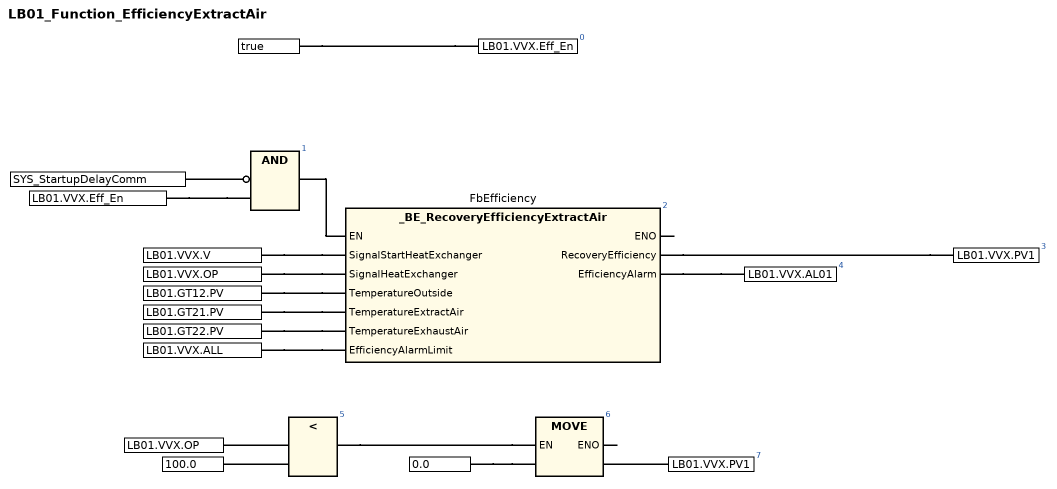
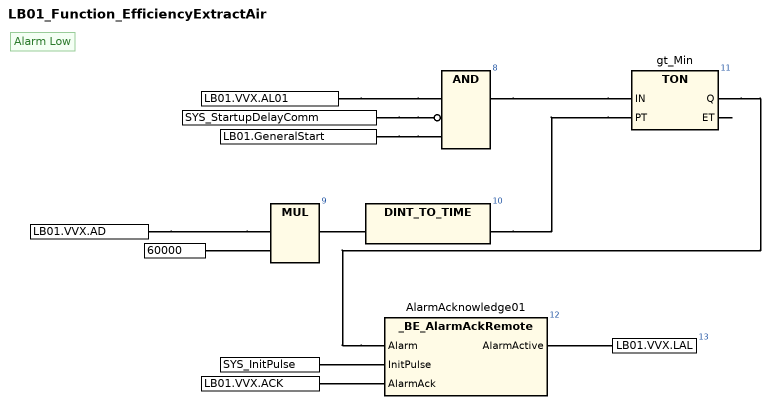
LB01.VVX.Eff_En := true;
IF NOT SYS_StartupDelayComm AND LB01.VVX.Eff_En THEN
    FbEfficiency(
        SignalStartHeatExchanger := LB01.VVX.V,
        SignalHeatExchanger := LB01.VVX.OP,
        TemperatureOutside := LB01.GT12.PV,
        TemperatureExtractAir := LB01.GT21.PV,
        TemperatureExhaustAir := LB01.GT22.PV,
        EfficiencyAlarmLimit := LB01.VVX.ALL); // _BE_RecoveryEfficiencyExtractAir
END_IF
LB01.VVX.PV1 := FbEfficiency.RecoveryEfficiency;
LB01.VVX.AL01 := FbEfficiency.EfficiencyAlarm;
IF LB01.VVX.OP < 100.0 THEN _w1 := 0.0; END_IF
LB01.VVX.PV1 := _w1;
// Alarm Low
gt_Min(IN := LB01.VVX.AL01 AND NOT SYS_StartupDelayComm AND LB01.GeneralStart, PT := DINT_TO_TIME(LB01.VVX.AD * 60000)); // TON
AlarmAcknowledge01(Alarm := gt_Min.Q, InitPulse := SYS_InitPulse, AlarmAck := LB01.VVX.ACK); // _BE_AlarmAckRemote
LB01.VVX.LAL := AlarmAcknowledge01.AlarmActive;

END_PROGRAM

// Device/AREA1/B001/LB01/Function/LB01_Function_Overtime
PROGRAM LB01_Function_Overtime
VAR
	FbOvertime: _BE_OverTime;
END_VAR

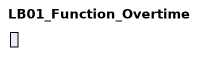
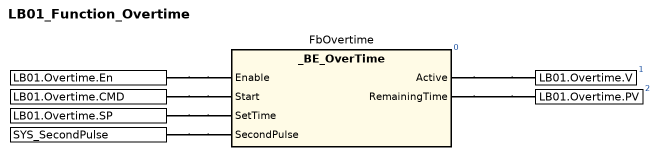
FbOvertime(
    Enable := LB01.Overtime.En,
    Start := LB01.Overtime.CMD,
    SetTime := LB01.Overtime.SP,
    SecondPulse := SYS_SecondPulse); // _BE_OverTime
LB01.Overtime.V := FbOvertime.Active;
LB01.Overtime.PV := FbOvertime.RemainingTime;

END_PROGRAM

// Device/AREA1/B001/LB01/Function/LB01_Function_Preheating
PROGRAM LB01_Function_Preheating
VAR
	plsGeneralStart: BOOL;
	plsStart: R_TRIG;
	delayStartControl: TON;
END_VAR
VAR // added by the converter: edge detectors and wires of the graphical bodies
    _w1, _w3, _w4 : ANY;
    _w2 : BOOL;
END_VAR

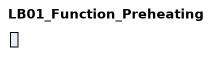
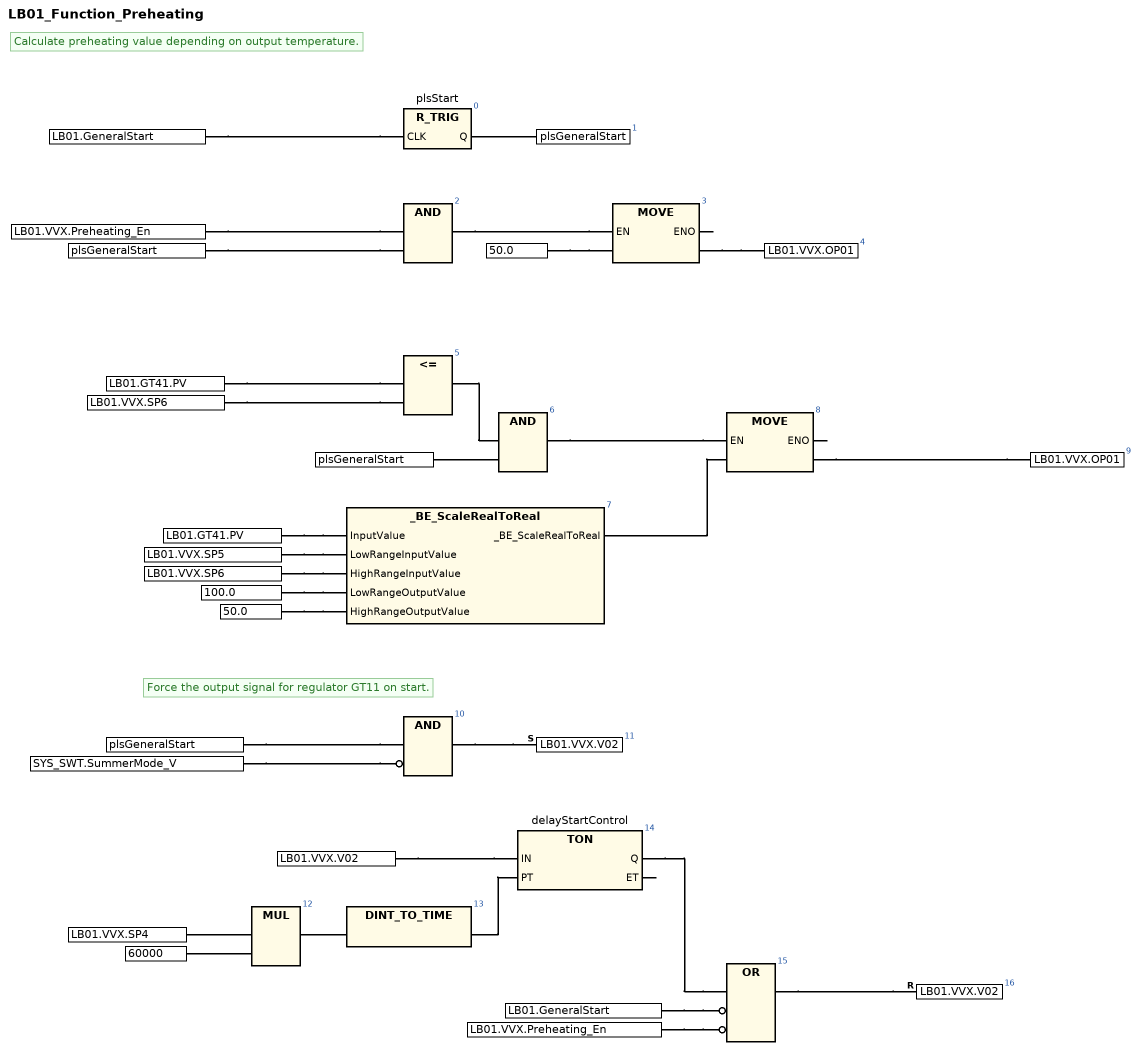
// Calculate preheating value depending on output temperature.
plsStart(CLK := LB01.GeneralStart); // R_TRIG
plsGeneralStart := plsStart.Q;
IF LB01.VVX.Preheating_En AND plsGeneralStart THEN _w1 := 50.0; END_IF
LB01.VVX.OP01 := _w1;
_w2 := LB01.GT41.PV <= LB01.VVX.SP6 AND plsGeneralStart;
_w3 := _BE_ScaleRealToReal(InputValue := LB01.GT41.PV, LowRangeInputValue := LB01.VVX.SP5, HighRangeInputValue := LB01.VVX.SP6, LowRangeOutputValue := 100.0, HighRangeOutputValue := 50.0);
IF _w2 THEN _w4 := _w3; END_IF
LB01.VVX.OP01 := _w4;
// Force the output signal for regulator GT11 on start.
LB01.VVX.V02 S= plsGeneralStart AND NOT SYS_SWT.SummerMode_V;
delayStartControl(IN := LB01.VVX.V02, PT := DINT_TO_TIME(LB01.VVX.SP4 * 60000)); // TON
LB01.VVX.V02 R= delayStartControl.Q OR NOT LB01.GeneralStart OR NOT LB01.VVX.Preheating_En;

END_PROGRAM

// Device/AREA1/B001/LB01/Sensor/Humidity/GM21/LB01_GM21
PROGRAM LB01_GM21
VAR
	local:strSensor7_Humidity;
	gt_Min: TON;
	gt_Max: TON;
	reset_en: RS;
	ackLal: BOOL;
	ackHal: BOOL;
	AlarmAcknowledge01: _BE_AlarmAckRemote;
	AlarmAcknowledge02: _BE_AlarmAckRemote;
END_VAR
VAR // added by the converter: edge detectors and wires of the graphical bodies
    _w1, _w3, _w4 : ANY;
    _w2 : BOOL;
END_VAR

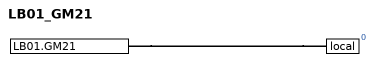
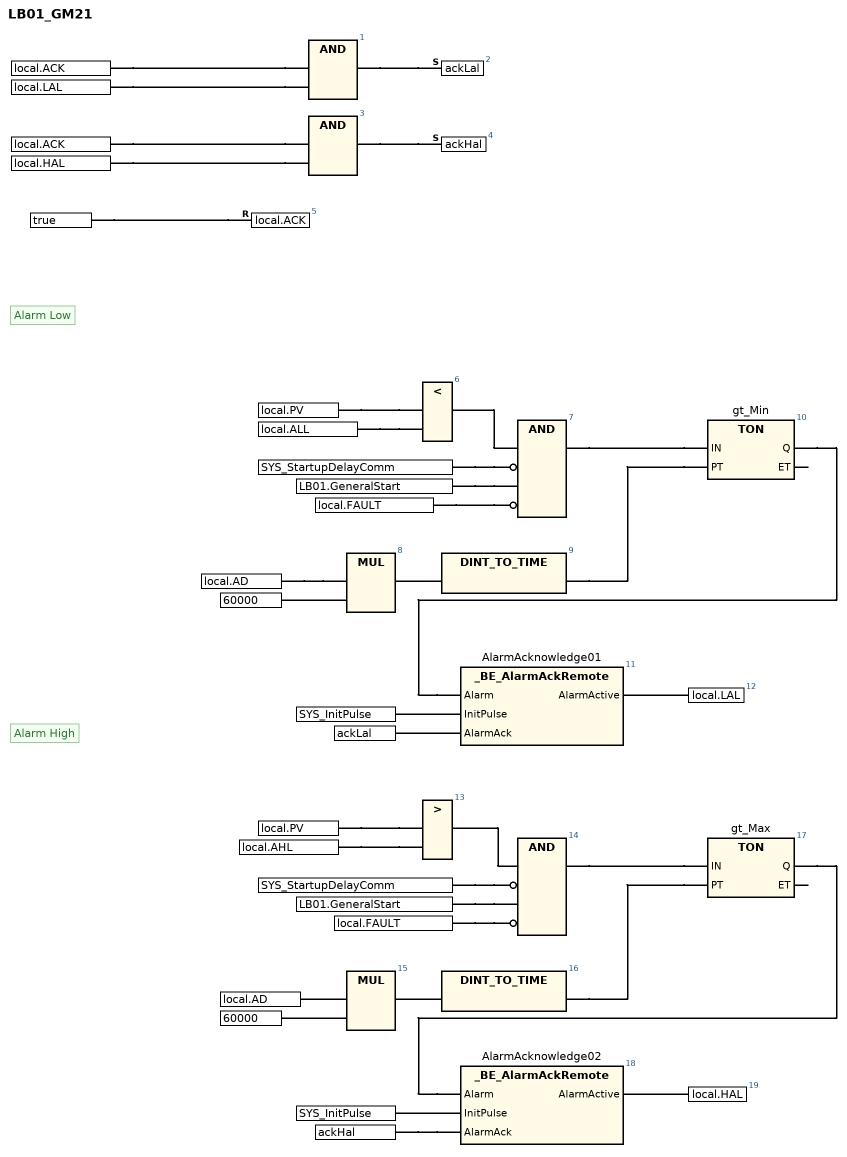
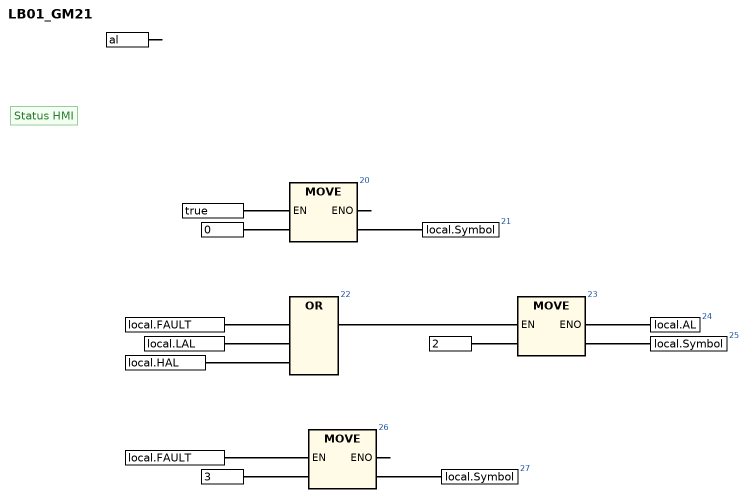
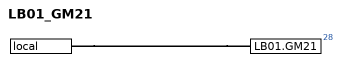
// note: 4 stored wires end on pins the file does not list and are not shown
local := LB01.GM21;
ackLal S= local.ACK AND local.LAL;
ackHal S= local.ACK AND local.HAL;
local.ACK R= true;
// Alarm Low
gt_Min(IN := local.PV < local.ALL AND NOT SYS_StartupDelayComm AND LB01.GeneralStart AND NOT local.FAULT, PT := DINT_TO_TIME(local.AD * 60000)); // TON
AlarmAcknowledge01(Alarm := gt_Min.Q, InitPulse := SYS_InitPulse, AlarmAck := ackLal); // _BE_AlarmAckRemote
local.LAL := AlarmAcknowledge01.AlarmActive;
// Alarm High
gt_Max(IN := local.PV > local.AHL AND NOT SYS_StartupDelayComm AND LB01.GeneralStart AND NOT local.FAULT, PT := DINT_TO_TIME(local.AD * 60000)); // TON
AlarmAcknowledge02(Alarm := gt_Max.Q, InitPulse := SYS_InitPulse, AlarmAck := ackHal); // _BE_AlarmAckRemote
local.HAL := AlarmAcknowledge02.AlarmActive;
// Status HMI
IF true THEN _w1 := 0; END_IF
local.Symbol := _w1;
_w2 := local.FAULT OR local.LAL OR local.HAL;
IF _w2 THEN _w3 := 2; END_IF
local.AL := _w2;
local.Symbol := _w3;
IF local.FAULT THEN _w4 := 3; END_IF
local.Symbol := _w4;
LB01.GM21 := local;
// al: input not connected

END_PROGRAM

// Device/AREA1/B001/LB01/Function/LB01_NightCooling
PROGRAM LB01_NightCooling
VAR
	fbNightCool: _BE_NightCooling;
END_VAR

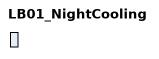
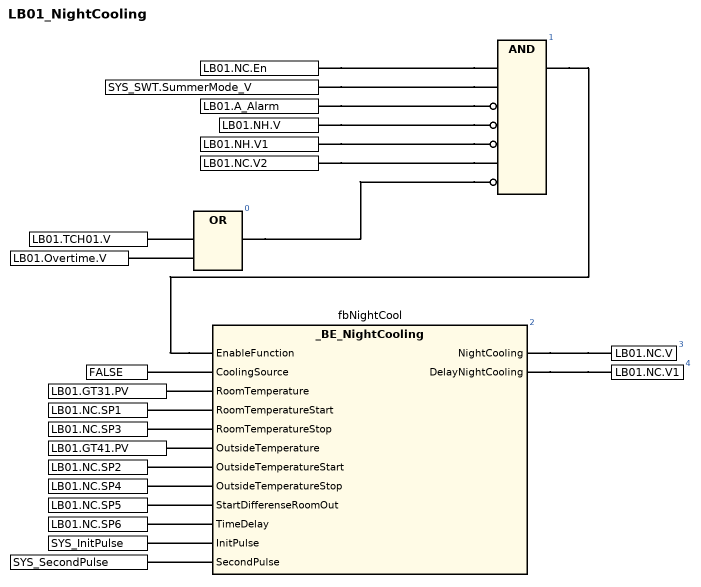
fbNightCool(
    EnableFunction := LB01.NC.En AND SYS_SWT.SummerMode_V AND NOT LB01.A_Alarm AND NOT LB01.NH.V AND NOT LB01.NH.V1 AND LB01.NC.V2 AND NOT (LB01.TCH01.V OR LB01.Overtime.V),
    CoolingSource := FALSE,
    RoomTemperature := LB01.GT31.PV,
    RoomTemperatureStart := LB01.NC.SP1,
    RoomTemperatureStop := LB01.NC.SP3,
    OutsideTemperature := LB01.GT41.PV,
    OutsideTemperatureStart := LB01.NC.SP2,
    OutsideTemperatureStop := LB01.NC.SP4,
    StartDifferenseRoomOut := LB01.NC.SP5,
    TimeDelay := LB01.NC.SP6,
    InitPulse := SYS_InitPulse,
    SecondPulse := SYS_SecondPulse); // _BE_NightCooling
LB01.NC.V := fbNightCool.NightCooling;
LB01.NC.V1 := fbNightCool.DelayNightCooling;

END_PROGRAM

// Device/AREA1/B001/LB01/Function/LB01_NightHeating
PROGRAM LB01_NightHeating
VAR
	fbNightHeat: _BE_NightHeating;
END_VAR

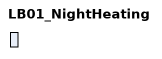
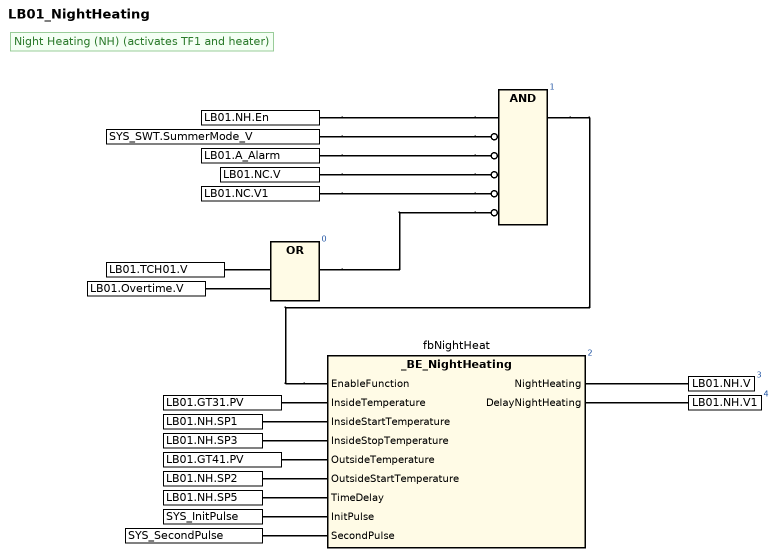
// Night Heating (NH) (activates TF1 and heater)
fbNightHeat(
    EnableFunction := LB01.NH.En AND NOT SYS_SWT.SummerMode_V AND NOT LB01.A_Alarm AND NOT LB01.NC.V AND NOT LB01.NC.V1 AND NOT (LB01.TCH01.V OR LB01.Overtime.V),
    InsideTemperature := LB01.GT31.PV,
    InsideStartTemperature := LB01.NH.SP1,
    InsideStopTemperature := LB01.NH.SP3,
    OutsideTemperature := LB01.GT41.PV,
    OutsideStartTemperature := LB01.NH.SP2,
    TimeDelay := LB01.NH.SP5,
    InitPulse := SYS_InitPulse,
    SecondPulse := SYS_SecondPulse); // _BE_NightHeating
LB01.NH.V := fbNightHeat.NightHeating;
LB01.NH.V1 := fbNightHeat.DelayNightHeating;

END_PROGRAM

// Device/AREA1/B001/UC/Sh1/Alarms/UCSh1_Alarms
PROGRAM UCSh1_Alarms
VAR
	AlarmAcknowledge01: _BE_AlarmAckRemote;
	timerManMode: TON;
	_BE_AlarmAckRemote_0: _BE_AlarmAckRemote;
END_VAR
VAR // added by the converter: edge detectors and wires of the graphical bodies
    _w1 : BOOL;
END_VAR

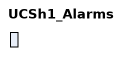
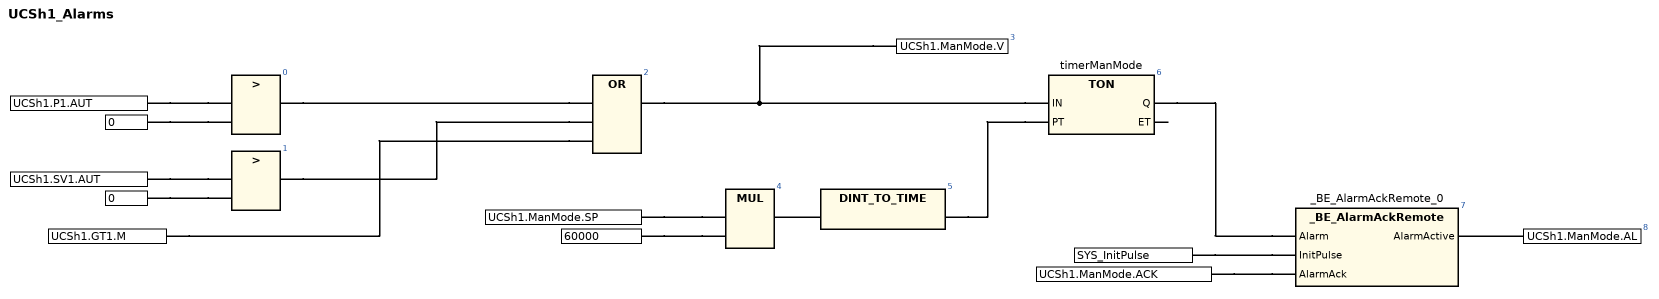
_w1 := UCSh1.P1.AUT > 0 OR UCSh1.SV1.AUT > 0 OR UCSh1.GT1.M;
UCSh1.ManMode.V := _w1;
timerManMode(IN := _w1, PT := DINT_TO_TIME(UCSh1.ManMode.SP * 60000)); // TON
_BE_AlarmAckRemote_0(Alarm := timerManMode.Q, InitPulse := SYS_InitPulse, AlarmAck := UCSh1.ManMode.ACK); // _BE_AlarmAckRemote
UCSh1.ManMode.AL := _BE_AlarmAckRemote_0.AlarmActive;

END_PROGRAM

// Device/AREA1/B001/UC/Sh1/UcUnit/UCSh1_StartConditions
PROGRAM UCSh1_StartConditions
VAR

END_VAR

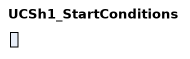
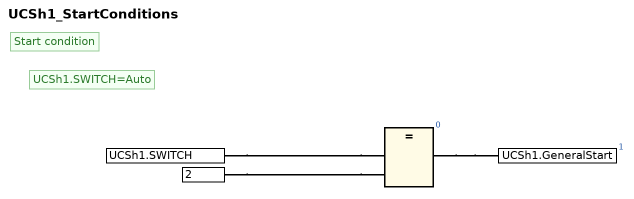
// Start condition
// UCSh1.SWITCH=Auto
UCSh1.GeneralStart := UCSh1.SWITCH = 2;

END_PROGRAM

// Device/AREA1/B001/UC/Sh1/Pump/UCSh1_P1
PROGRAM UCSh1_P1
VAR
	local:strPumpExercise;
	fbControlPump2: _BE_Pump_2;
	fbPumpStartCondition: _BE_PumpStartConditions;
	fb_OperationalTime: _BE_OperationalTime;
	fbExercise: _BE_Exercise;
	ackAl01: BOOL;
	ackAl02: BOOL;
	sv_op: REAL;
	startPump: BOOL;
	AlarmFb01: _BE_AlarmAckRequired;
	AlarmFb02: _BE_AlarmAckRequired;
END_VAR
VAR // added by the converter: edge detectors and wires of the graphical bodies
    _w1 : ANY;
END_VAR

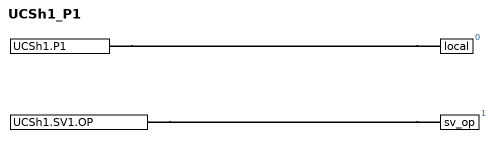
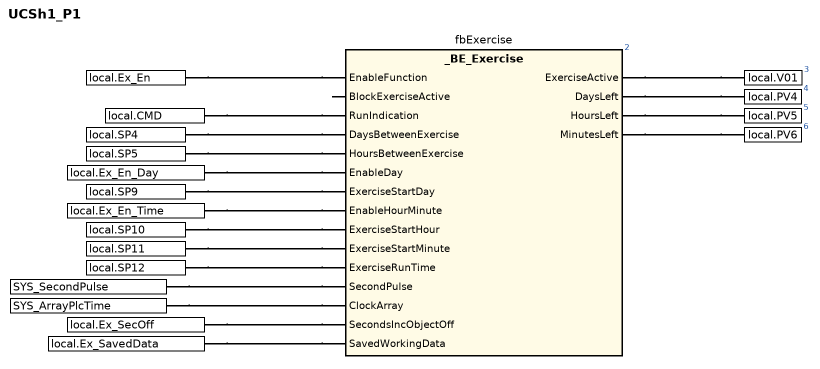
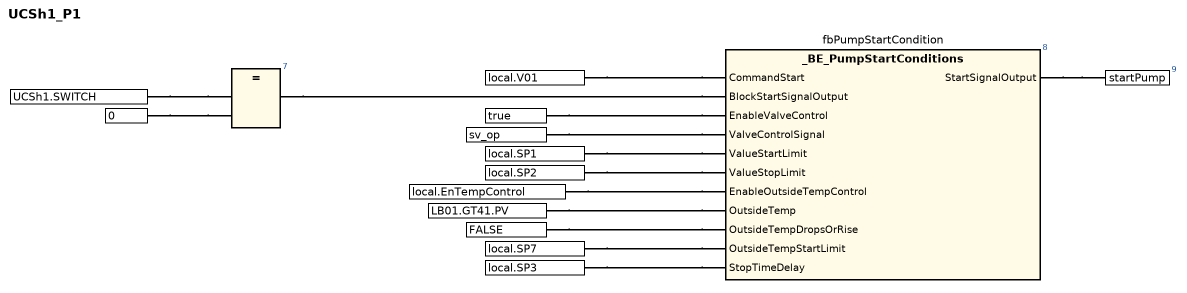
